{attribute addProperty BoxType "AT2050-0501-0022"}
{attribute addProperty Id "A_0082_AT2002_5250_0019_AT2002_5250AT2002_3DCFC8D064080"}
{attribute addProperty CRC "597683380"}
{attribute addProperty SizeInBites "640"}
{attribute addProperty SizeInBytes "80"}
TYPE A_0070_AT2050_0501_0022_AT2050_0501_239FECB4 EXTENDS AT2050_9506A482 :
STRUCT
	{attribute addProperty Name "A_0082_AT2002_5250_0019_AT2002_5250"}
	A_0082_AT2002_5250_0019_AT2002_5250 : AT2002_3DCFC8D0;
END_STRUCT
END_TYPE

(* stored: Version 1.2.0.0, ProductVersion 3.1.4024.9
   DUT A_0070_AT2050_0501_0022_AT2050_0501_239FECB4: Id {bdf3cdd3-b28c-40e8-b67e-a67ee30f5f58} *)
